PROGRAM MAIN
VAR
	jsonDomParser_TestSuit : JsonDomParser_TestSuit;
END_VAR

TcUnit.RUN();

END_PROGRAM

(* stored: Version 1.1.0.1, ProductVersion 3.1.4024.12
   POU MAIN: Id {571dcd2b-7f1a-0119-09ce-d4765fa24bb1}, SpecialFunc None *)
